PROGRAM MAIN
VAR
END_VAR

Orderverwerking_magazijn ();
Transporteren_order();

END_PROGRAM

(* stored: Version 1.1.0.1, ProductVersion 3.1.4024.12
   POU MAIN: Id {e7b53381-7db3-4f45-a7b7-c24bd15252a5}, SpecialFunc None *)
